// TIA Portal V19 export
DATA_BLOCK "A0304_Navetta"   // DB6
// stored: InstanceOfName A0304_Navetta_FB, InstanceOfType FB
"A0304_Navetta_FB"
   // VAR_INPUT
   //    AreaInterface : "AreaInterface";
   //    ZSI : "udt_ZoneSafetyInterface";
   //    DSI_Feed_Testa : "udt_DeviceSafetyInterface";
   //    DSI_Feed_Coda : "udt_DeviceSafetyInterface";
   //    DSI_Valve : "udt_DeviceSafetyInterface";
   //    DataIn : Struct
   //       OP_Vai_A_Prelievo : Bool;
   //       OP_Vai_A_Deposito : Bool;
   //       OP_Prelievo : Bool;
   //       OP_Deposito : Bool;
   //       UnloadBenchCaricoMatPres1 : Bool;
   //       UnloadBenchCaricoMatPres2 : Bool;
   //       UnloadBenchScaricoMatPres1 : Bool;
   //       UnloadBenchScaricoMatPres2 : Bool;
   //       PalettoInternoCoda_LsRest : Bool;
   //       PalettoInternoCoda_LsWork : Bool;
   //       PalettoInternoTesta_LsRest : Bool;
   //       PalettoInternoTesta_LsWork : Bool;
   //       PalettoEsternoCoda_LsRest : Bool;
   //       PalettoEsternoCoda_LsWork : Bool;
   //       PalettoEsternoTesta_LsRest : Bool;
   //       PalettoEsternoTesta_LsWork : Bool;
   //    END_STRUCT;
   //    CIn : Struct
   //       Manager : Struct
   //          EnableStopDoorOpeningReq : Bool;
   //          EnableStopInPhase : Bool;
   //          EnableStopProgrammed : Bool;
   //          Control_ON : Bool;
   //          CanMoveFreely { ExternalAccessible := 'False'; ExternalVisible := 'False'; ExternalWritable := 'False'} : Bool;
   //          Phase : Struct
   //             VAI_A_PRELIEVO : Bool;
   //             PRELIEVO : Bool;
   //             VAI_A_DEPOSITO : Bool;
   //             DEPOSITO : Bool;
   //          END_STRUCT;
   //       END_STRUCT;
   //       Sostegno : Struct
   //          ReadyForDeposito : Bool;
   //       END_STRUCT;
   //       Sollevatori : Struct
   //          Testa : Struct
   //             InPosDeposito : Bool;
   //             ActualPos : LReal;
   //          END_STRUCT;
   //          Coda : Struct
   //             InPosDeposito : Bool;
   //             ActualPos : LReal;
   //          END_STRUCT;
   //       END_STRUCT;
   //       AirOk : Bool;
   //       CycleModeShortPiece : Bool;
   //    END_STRUCT;
   //    Config : Struct
   //       Navetta : Struct
   //          Testa : Struct
   //             Ax : "Positioning_DOL_Machine_Config";
   //             PalettiEsterni : "ValveMachine_Config";
   //             PalettiInterni : "ValveMachine_Config";
   //          END_STRUCT;
   //          Coda : Struct
   //             Ax : "Positioning_DOL_Machine_Config";
   //             PalettiEsterni : "ValveMachine_Config";
   //             PalettiInterni : "ValveMachine_Config";
   //          END_STRUCT;
   //          DelayMissingCondition { ExternalAccessible := 'False'; ExternalVisible := 'False'; ExternalWritable := 'False'} : Time;
   //       END_STRUCT;
   //    END_STRUCT;
   // END_VAR
   // VAR_OUTPUT
   //    MachineInterface : "MachineInterface";
   //    COut : Struct
   //       Testa : Struct
   //          Ax : "Positioning_DOL_Machine_COut";
   //          PalettiEsterni : "ValveMachine_COut";
   //          PalettiInterni : "ValveMachine_COut";
   //       END_STRUCT;
   //       Coda : Struct
   //          Ax : "Positioning_DOL_Machine_COut";
   //          PalettiEsterni : "ValveMachine_COut";
   //          PalettiInterni : "ValveMachine_COut";
   //       END_STRUCT;
   //       Cumulativo : Struct
   //          PalettiEsterni : "ValveMachine_COut";
   //          PalettiInterni : "ValveMachine_COut";
   //       END_STRUCT;
   //       ReadyToRecive : Bool;
   //    END_STRUCT;
   //    DataOut : Struct
   //       Testa : Struct
   //          PalettoEsterno : Struct
   //             SbloccaggioStelo : Bool;
   //             Rest : Bool;
   //             Work : Bool;
   //          END_STRUCT;
   //          PalettoInterno : Struct
   //             SbloccaggioStelo : Bool;
   //             Rest : Bool;
   //             Work : Bool;
   //          END_STRUCT;
   //       END_STRUCT;
   //       Coda : Struct
   //          PalettoEsterno : Struct
   //             SbloccaggioStelo : Bool;
   //             Rest : Bool;
   //             Work : Bool;
   //          END_STRUCT;
   //          PalettoInterno : Struct
   //             SbloccaggioStelo : Bool;
   //             Rest : Bool;
   //             Work : Bool;
   //          END_STRUCT;
   //       END_STRUCT;
   //    END_STRUCT;
   // END_VAR
   // VAR_IN_OUT
   //    Par : Struct
   //       Ax_Man : "Positioning_DOL_Machine_Par";
   //       Ax_Testa_Pers : "Positioning_DOL_Machine_Pers_Data";
   //       Ax_Coda_Pers : "Positioning_DOL_Machine_Pers_Data";
   //       Enc : Struct
   //          Testa : "PosFbk_RTN";
   //          Coda : "PosFbk_RTN";
   //       END_STRUCT;
   //    END_STRUCT;
   //    Par_Mach : Struct
   //       PosPrePrelievo : LReal;
   //       PosPrelievo : LReal;
   //       PosDeposito : LReal;
   //       ToleranceWindow : LReal;
   //    END_STRUCT;
   // END_VAR
   // VAR
   //    Alarm : Struct
   //       Testa : Struct
   //          Ax : "Positioning_DOL_Machine_Alr";
   //          Enc : "PosFbk_Encoder_Alr";
   //          PalettiEsterni : "ValveAlr";
   //          PalettiInterni : "ValveAlr";
   //       END_STRUCT;
   //       Coda : Struct
   //          Ax : "Positioning_DOL_Machine_Alr";
   //          Enc : "PosFbk_Encoder_Alr";
   //          PalettiEsterni : "ValveAlr";
   //          PalettiInterni : "ValveAlr";
   //       END_STRUCT;
   //       CheckBothShutMove : Bool;
   //    END_STRUCT;
   //    Warning : Struct
   //       Testa : Struct
   //          Ax { S7_SetPoint := 'True'} : "Positioning_DOL_Machine_Wng";
   //          PalettiEsterni : "ValveMachine_Wng";
   //          PalettiInterni : "ValveMachine_Wng";
   //       END_STRUCT;
   //       Coda : Struct
   //          Ax { S7_SetPoint := 'True'} : "Positioning_DOL_Machine_Wng";
   //          PalettiEsterni : "ValveMachine_Wng";
   //          PalettiInterni : "ValveMachine_Wng";
   //       END_STRUCT;
   //       MissingCnd : Struct
   //          OP_VAI_A_PRELIEVO : Bool;
   //          OP_PRELIEVO : Bool;
   //          OP_VAI_A_DEPOSITO : Bool;
   //          OP_DEPOSITO : Bool;
   //       END_STRUCT;
   //    END_STRUCT;
   //    HMI : Struct
   //       Selection : Struct
   //          Ax : Int;
   //          PalettiEsterni : Int;
   //          PalettiInterni : Int;
   //       END_STRUCT;
   //       Testa : Struct
   //          PbPreset : Bool;
   //          PresetValue : LReal;
   //       END_STRUCT;
   //       Coda : Struct
   //          PbPreset : Bool;
   //          PresetValue : LReal;
   //       END_STRUCT;
   //    END_STRUCT;
   //    Sts : Struct
   //       OP_CanMoveFreely : Bool;
   //       OP_Vai_A_Prelievo_Cnd : Bool;
   //       OP_Prelievo_Cnd : Bool;
   //       OP_Vai_A_Deposito_Cnd : Bool;
   //       OP_Deposito_Cnd : Bool;
   //       Coda_PermessoDaSynchOk : Bool;
   //       Testa_PermessoDaSynchOk : Bool;
   //       OutOfWorkSpace : Bool;
   //       GenCndFwd : Bool;
   //       GenCndBkw : Bool;
   //       ReloadAirRequest : Bool;
   //       InPosPrelievo : Bool;
   //       InPosPrePrelievo : Bool;
   //       InPosDeposito : Bool;
   //    END_STRUCT;
   //    Ctrl : Struct
   //       Man : Struct
   //          OP_Vai_A_Prelievo : Bool;
   //          OP_Prelievo : Bool;
   //          OP_Vai_A_Deposito : Bool;
   //          OP_Deposito : Bool;
   //       END_STRUCT;
   //       Aut : Struct
   //          OP_Vai_A_Prelievo : Bool;
   //          OP_Prelievo : Bool;
   //          OP_Vai_A_Deposito : Bool;
   //          OP_Deposito : Bool;
   //       END_STRUCT;
   //       OP_Vai_A_Prelievo : Bool;
   //       OP_Prelievo : Bool;
   //       OP_Vai_A_Deposito : Bool;
   //       OP_Deposito : Bool;
   //       ReloadAir { S7_SetPoint := 'True'} : Bool;
   //    END_STRUCT;
   //    Ax_Testa { S7_SetPoint := 'True'} : "Positioning_DOL_Machine_FB";
   //    Ax_Coda { S7_SetPoint := 'True'} : "Positioning_DOL_Machine_FB";
   //    PalettiEsterni_Testa { S7_SetPoint := 'True'} : "ValveMachine_FB";
   //    PalettiEsterni_Coda { S7_SetPoint := 'True'} : "ValveMachine_FB";
   //    PalettiInterni_Testa { S7_SetPoint := 'True'} : "ValveMachine_FB";
   //    PalettiInterni_Coda { S7_SetPoint := 'True'} : "ValveMachine_FB";
   //    BloccaggioStelo_PalettoEsterno_Testa { S7_SetPoint := 'True'} : "Valve";
   //    BloccaggioStelo_PalettoEsterno_Coda { S7_SetPoint := 'True'} : "Valve";
   //    Enc_Testa : "PosFbk_SickAFM60";
   //    Enc_Testa_ITF : "PosFbk_ITF";
   //    Enc_Coda : "PosFbk_SickAFM60";
   //    Enc_Coda_ITF : "PosFbk_ITF";
   //    AUX { ExternalAccessible := 'False'; ExternalVisible := 'False'; ExternalWritable := 'False'} : Struct
   //       OP_Vai_A_Prelievo : Bool;
   //       OP_Prelievo : Bool;
   //       OP_Vai_A_Deposito : Bool;
   //       OP_Deposito : Bool;
   //       AirOk : Bool;
   //       Clock250 : Bool;
   //    END_STRUCT;
   //    TON_OP_VAI_A_PRELIEVO_MissingCnd : IEC_TIMER;
   //    TON_OP_PRELIEVO_MissingCnd : IEC_TIMER;
   //    TON_OP_VAI_A_DEPOSITO_MissingCnd : IEC_TIMER;
   //    TON_OP_DEPOSITO_MissingCnd : IEC_TIMER;
   //    TON_CheckShuttleMove { S7_SetPoint := 'True'} : IEC_TIMER;
   //    TON_ReloadAir { S7_SetPoint := 'True'} : IEC_TIMER;
   //    TON_CheckAxis { S7_SetPoint := 'True'} : IEC_TIMER;
   //    CheckAxisSynch { ExternalAccessible := 'False'; ExternalVisible := 'False'; ExternalWritable := 'False'} : "CheckAxisSynch";
   //    Sts_PosAxis { S7_SetPoint := 'True'} : Int;
   // END_VAR
BEGIN
END_DATA_BLOCK
